Fanuc KAREL source: GET_JPOS_TPE.kl

PROGRAM T
%NOLOCKGROUP
VAR
 v0 : INTEGER
 v1 : INTEGER
 v2 : INTEGER
 v3 : INTEGER
 res : JOINTPOS
BEGIN
 res = GET_JPOS_TPE(v0, v1, v2, v3)
END T
